(* PLC project 117_1_V0.5.project, CODESYS CODESYS V3.5 SP17 Patch 3 *)
(* stored: creationDateTime 1970-01-01T00:00:00, modificationDateTime 2026-06-16T22:51:19.9979415 *)

{attribute 'strict'}
TYPE STATUS : (NOT_COMMUNICATION, OFF, READY, MOVING, ERROR);
END_TYPE
